{attribute 'qualified_only'}
VAR_GLOBAL
END_VAR

(* stored: Version 1.1.0.1, ProductVersion 3.1.4024.13
   GVL GVL_EIP: Id {c78af690-db02-4775-b2cb-37f8f9a201b8} *)
